// TwinCAT 3 PLC project zaverecne_zadanie
// ProgramVersion: 3.1.4024.0
// libraries:
//   Tc2_Standard, * (Beckhoff Automation GmbH)
//   Tc2_System, * (Beckhoff Automation GmbH)
//   Tc3_Module, * (Beckhoff Automation GmbH)
// project tree:
//   / PlcTask.TcTTO
//   POUs/ MAIN.TcPOU, zadanie_zapocet.TcPOU
// real-time tasks:
//   TASK PlcTask: cycle T#10ms, priority 20, ADS port 350

CONFIGURATION zaverecne_zadanie
    RESOURCE PLC ON TwinCAT3
        TASK PlcTask(INTERVAL := T#10ms, PRIORITY := 20);
        PROGRAM MAIN WITH PlcTask : MAIN;
        PROGRAM zadanie_zapocet WITH PlcTask : zadanie_zapocet;
    END_RESOURCE
END_CONFIGURATION

// ---- POUs/MAIN.TcPOU
PROGRAM MAIN
VAR
END_VAR

END_PROGRAM

// ---- POUs/zadanie_zapocet.TcPOU
PROGRAM zadanie_zapocet
VAR
	M1: BOOL;
	M2: BOOL;
	M3: BOOL;
	start: BOOL;
	stop1: BOOL;
	stav: UINT;
	stop2: BOOL;
	stop3: BOOL;
	casovac: TON;
END_VAR

CASE stav OF 
	0: M1 := FALSE; 
	   M2 := FALSE; 
	   M3 := FALSE; 
	   casovac.IN := FALSE; 
	   casovac(); 
	IF start = TRUE THEN
		stav := 10; 
	END_IF
	10: M1 := TRUE; 
		M2 := FALSE; 
		M3 := FALSE; 
		casovac.IN := TRUE; 
		casovac.PT := T#5S; 
		casovac(); 
		IF casovac.Q = TRUE THEN
			stav := 20; 
		END_IF
		
	20: M1 := TRUE;
		M2 := TRUE;
		M3 := TRUE;
	IF stop1 = TRUE THEN 
		stav := 30;
		END_IF
	30: M1 := FALSE;
		M2 := TRUE;
		M3 := TRUE;
	IF stop3 = TRUE THEN 
		stav := 40;
	END_IF
	40: M1 := FALSE;
		M2 := TRUE;
		M3 := FALSE;
	IF stop2 = TRUE THEN 
		stav := 50;
	END_IF
	50: M1 := FALSE;
		M2 := FALSE;
		M3 := FALSE;
END_CASE

END_PROGRAM
